Staubli VAL3: save.pgx

public program save(string x_sName, num& x_nResult[])
begin
  // save it
  if isDefined(saveProg:pProg[pEdit.sID])
    saveProg:pProg[pEdit.sID]=pEdit
  endIf
  x_nResult=saveProg:libSave()
end
